// TIA Portal V20 export
FUNCTION_BLOCK "RealFbName2"   // FB3, LAD
   VAR CONSTANT
      MaxSpeedError : Int := 50;
      MinSpeed : Real := 20.0;
   END_VAR
BEGIN
END_FUNCTION_BLOCK
